RoboDK station: TRABAJO PRACTICO 7.rdk

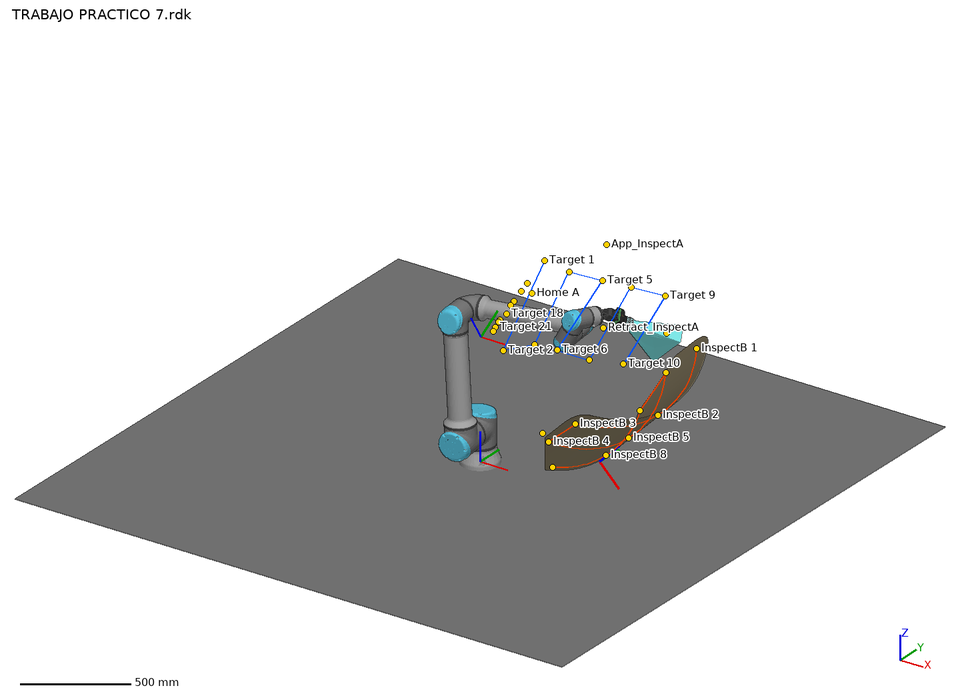
[picture v0: the station drawn from its stored meshes, robots at their saved joint values, targets as dots, program paths as lines]
Station TRABAJO PRACTICO 5 (saved by RoboDK 5.7.2). Poses are relative to the parent item; angles as X-Y-Z fixed-axis rotations.
Station parameters (name, value as stored): Palletizing Plugin
  - frame UR10e Base at (0, 0, 0) mm
    - robot UR10e: 6 axes, payload 10 kg, reach 1300 mm, repeatability 0.05 mm, weight 28.9 kg
        modified DH rows (alpha deg, a mm, theta deg, d mm): 0, 0, 0, 180.7; 90, 0, 180, 0; 0, 612.6, 0, 0; 0, 571.335, 0, 174.15; -90, 0, 0, 119.85; 90, 0, 180, 116.55
        joint limits [-360, -360, -360, -360, -360, -360] to [360, 360, 360, 360, 360, 360]; home [0, -90, -90, 0, 90, 0]; saved at [6.14, -86.815, -90.402, -30.486, 158.848, 109.654]
      - tool Camera 2, TCP at (0, -175.95, 321.06) mm, rotated rx 40 ry 0 rz 0 deg, size 215.7 x 276.1 x 372.4 mm
  - frame Frame Inspection A at (-380.72, 553.59, 295.24) mm, rotated rx 32.84 ry 0 rz 0 deg
    - object Inspection A at (0, 0, 0) mm, size 800 x 500 x 0 mm, geometry from Inspection A.step
    - folder TargetsA
    - target Target 1 (Cartesian target) at (79.2, 457.51, 5) mm, rotated rx -180 ry 0 rz 180 deg; joints [133.501, -90.589, -95.318, -17.151, 48.873, 195.641] of UR10e
    - target Target 2 (Cartesian target) at (141.75, -34.27, 5) mm, rotated rx 179.75 ry 0 rz 180 deg; joints [184.834, -41.161, -136.372, -107.963, 17.565, 286.215] of UR10e
    - target Target 3 (Cartesian target) at (270.26, 41.79, 5) mm, rotated rx 180 ry 0 rz 180 deg; joints [161.24, -38.764, -144.388, -40.681, 25.213, 220.978] of UR10e
    - target Target 4 (Cartesian target) at (224.75, 441.5, 5) mm, rotated rx -180 ry 0 rz 180 deg; joints [123.151, -84.661, -102.076, -13.507, 58.499, 190.907] of UR10e
    - target Target 5 (Cartesian target) at (403.61, 448.09, 5) mm, rotated rx -180 ry 0 rz 180 deg; joints [105.682, -83.563, -102.861, -11.357, 75.033, 184.735] of UR10e
    - target Target 6 (Cartesian target) at (390.7, 47.14, 5) mm, rotated rx 180 ry 0 rz 180 deg; joints [137.831, -39.235, -146.275, -19.19, 44.913, 198.041] of UR10e
    - target Target 7 (Cartesian target) at (568.48, 46.93, 5) mm, rotated rx -180 ry 0 rz 180 deg; joints [86.626, -56.24, -142.379, 1.432, 93.224, 179.004] of UR10e
    - target Target 8 (Cartesian target) at (554.74, 458.13, 5) mm, rotated rx -180 ry 0 rz 180 deg; joints [90.013, -86.994, -99.225, -10.94, 89.988, 180.004] of UR10e
    - target Target 9 (Cartesian target) at (750.45, 458.08, 25) mm, rotated rx 180 ry 0 rz 180 deg; joints [71.618, -93.897, -90.519, -13.607, 107.537, 174.401] of UR10e
    - target Target 10 (Cartesian target) at (750.21, 68.01, 25) mm, rotated rx 180 ry 0 rz 180 deg; joints [55.701, -74.55, -129.53, 3.586, 122.577, 168.622] of UR10e
    - target App_InspectA (Cartesian target) at (433.96, 543.11, 175.01) mm, rotated rx -172.24 ry 18.28 rz 174.82 deg; joints [115.29, -89.41, -72.94, -49.41, 49.41, 188.24] of UR10e
    - target Retract_InspectA (Cartesian target) at (750.21, 68.01, 315) mm, rotated rx 180 ry 0 rz -180 deg; joints [39.031, -62.165, -111.409, -32.544, 137.922, 160.003] of UR10e
    - target Home A (joint target) at (558.33, -45.25, 667.51) mm, rotated rx -180 ry 0 rz -180 deg; joints [90.932, -32.458, -85.483, -79.221, 89.109, 180.275] of UR10e
    - target Target 14 (Cartesian target) at (65.12, 323.89, 5) mm, rotated rx 180 ry 0 rz 179.79 deg; joints [142.957, -81.972, -110.313, -14.929, 40.175, 201.57] of UR10e
    - target Target 15 (Cartesian target) at (61.03, 276.19, 5) mm, rotated rx 180 ry 0 rz 179.79 deg; joints [146.894, -78.963, -115.197, -15.414, 36.711, 204.58] of UR10e
    - target Target 16 (Cartesian target) at (54.59, 218.09, 5) mm, rotated rx 180 ry 0 rz 179.79 deg; joints [152.333, -75.295, -120.754, -17.699, 32.077, 209.635] of UR10e
    - target Target 17 (Cartesian target) at (48.84, 192.68, 5) mm, rotated rx 180 ry 0 rz 179.79 deg; joints [155.072, -73.816, -122.904, -19.652, 29.834, 212.694] of UR10e
    - target Target 18 (Cartesian target) at (54.37, 146.46, 5) mm, rotated rx -180 ry -0.47 rz 179.79 deg; joints [159.377, -69.627, -127.627, -23.673, 26.763, 218.279] of UR10e
    - target Target 19 (Cartesian target) at (41.82, 108.93, 5) mm, rotated rx 180 ry 0 rz 179.79 deg; joints [164.318, -67.471, -129.772, -31.808, 22.992, 226.811] of UR10e
    - target Target 20 (Cartesian target) at (40.49, 96.72, 5) mm, rotated rx 180 ry 0 rz 179.79 deg; joints [165.792, -66.439, -130.582, -34.771, 22.053, 229.778] of UR10e
    - target Target 21 (Cartesian target) at (41.12, 65.11, 5) mm, rotated rx -180 ry 0 rz 179.79 deg; joints [169.618, -63.229, -132.561, -44.277, 19.903, 238.637] of UR10e
    - target Target 22 (Cartesian target) at (42.77, 42.7, 5) mm, rotated rx -180 ry 0 rz 179.79 deg; joints [172.451, -60.718, -133.61, -53.008, 18.646, 246.336] of UR10e
  - frame Frame Inspection B at (727.24, -100, 245.26) mm, rotated rx 0 ry 45.31 rz 0 deg
    - object Inspection B at (0, 0, 0) mm, size 202.5 x 1023.2 x 500 mm, geometry from Inspection B.step
    - target InspectB 1 (Cartesian target) at (-169.52, 507.12, 414.46) mm, rotated rx 90.86 ry 88.34 rz 129.57 deg; joints [15.023, -98.718, -87.565, -11.255, 155.215, 119.931] of UR10e
    - target InspectB 2 (Cartesian target) at (-6.3, 34.85, 422.21) mm, rotated rx 90 ry 88.73 rz 89.24 deg; joints [-2.551, -95.184, -85.812, -44.784, 131.035, 89.277] of UR10e
    - target InspectB 3 (Cartesian target) at (-170.32, -428.18, 402.32) mm, rotated rx 89.84 ry 89 rz 51.46 deg; joints [-17.421, -91.076, -80.259, -55.032, 103.875, 78.266] of UR10e
    - target InspectB 4 (Cartesian target) at (-180.94, -441.02, 219.27) mm, rotated rx 91.56 ry 89 rz 52.19 deg; joints [-22.212, -79.982, -102.696, -44.394, 106.19, 74.724] of UR10e
    - target InspectB 5 (Cartesian target) at (-6.33, 32.62, 194.61) mm, rotated rx 90 ry 89.2 rz 89.24 deg; joints [-3.525, -82.536, -114.24, -30.023, 131.7, 87.717] of UR10e
    - target InspectB 6 (Cartesian target) at (-168.47, 505.6, 180.05) mm, rotated rx 93.22 ry 89.38 rz 132.09 deg; joints [19.329, -87.442, -116.77, 8.038, 151.578, 120.916] of UR10e
    - target InspectB 7 (Cartesian target) at (-96.46, 396.52, 16.99) mm, rotated rx 90.7 ry 89.4 rz 119.27 deg; joints [17.027, -80.228, -135.951, 10.169, 144.428, 112.006] of UR10e
    - target InspectB 8 (Cartesian target) at (-6.25, 41.26, 15.39) mm, rotated rx 90.07 ry 89.47 rz 90.84 deg; joints [-4.974, -75.499, -133.485, -19.186, 134.195, 85.804] of UR10e
    - target InspectB 9 (Cartesian target) at (-88.51, -301.4, 19.49) mm, rotated rx 90.88 ry 89.53 rz 63.85 deg; joints [-21.86, -72.359, -126.788, -31.965, 117.705, 73.128] of UR10e
    - target App_InspectB (Cartesian target) at (-298.16, 404, 414.54) mm, rotated rx 90.86 ry 88.34 rz 129.57 deg; joints [7.716, -89.072, -88.225, -26.91, 162.055, 112.785] of UR10e
    - target Retract_InspectB (Cartesian target) at (-242.37, -222.92, 19.51) mm, rotated rx 90.88 ry 89.53 rz 63.85 deg; joints [-15.839, -53.956, -125.352, -49.575, 113.831, 78.249] of UR10e
  - frame World at (0, 0, 0) mm
    - object Floor at (0, 0, -7) mm, size 3000 x 3000 x 4.2 mm, geometry from Floor.step
  - folder InspectA
    - program GoHomeA (3 instructions, listed below)
    - program InspectA (12 instructions, listed below)
    - program MainInspectA (5 instructions, listed below)
    - program App_InspectA (3 instructions, listed below)
    - program Retract_InspectA (3 instructions, listed below)
  - folder InspectB
    - program InspectB (8 instructions, listed below)
    - program App_InspectB (3 instructions, listed below)
    - program Retract_InspectB (3 instructions, listed below)
    - program Main_InspectB (3 instructions, listed below)
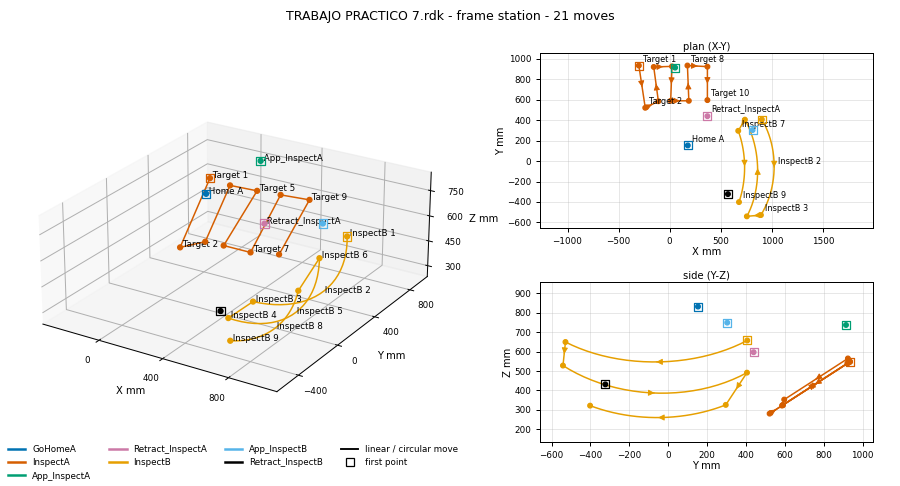
[picture p0: tool path of TRABAJO PRACTICO 7.rdk in frame station, 21 of 21 moves have a stored position in this frame; points joined in program order, loops and branches not executed]

--- program GoHomeA (robot UR10e) ---
  Est. Ref.: Frame Inspection A
  Est. herr: Camera 2
  MoveJ (Home A)

--- program InspectA (robot UR10e) ---
  Est. Ref.: Frame Inspection A
  Est. herr: Camera 2
  MoveJ (Target 1)
  MoveL (Target 2)
  MoveL (Target 3)
  MoveL (Target 4)
  MoveL (Target 5)
  MoveL (Target 6)
  MoveL (Target 7)
  MoveL (Target 8)
  MoveL (Target 9)
  MoveL (Target 10)

--- program MainInspectA (robot UR10e) ---
  Llamar GoHomeA
  Llamar App_InspectA
  Llamar InspectA
  Llamar Retract_InspectA
  Llamar GoHomeA

--- program App_InspectA (robot UR10e) ---
  Est. Ref.: Frame Inspection A
  Est. herr: Camera 2
  MoveJ (App_InspectA)

--- program Retract_InspectA (robot UR10e) ---
  Est. Ref.: Frame Inspection A
  Est. herr: Camera 2
  MoveL (Retract_InspectA)

--- program InspectB (robot UR10e) ---
  Est. Ref.: Frame Inspection B
  Est. herr: Camera 2
  MoveL (InspectB 1)
  MoveC (InspectB 2, InspectB 3)
  MoveL (InspectB 4)
  MoveC (InspectB 5, InspectB 6)
  MoveL (InspectB 7)
  MoveC (InspectB 8, InspectB 9)

--- program App_InspectB (robot UR10e) ---
  Est. Ref.: Frame Inspection B
  Est. herr: Camera 2
  MoveJ (App_InspectB)

--- program Retract_InspectB (robot UR10e) ---
  Est. Ref.: Frame Inspection B
  Est. herr: Camera 2
  MoveJ (Retract_InspectB)

--- program Main_InspectB (robot UR10e) ---
  Llamar App_InspectB
  Llamar Prog6
  Llamar Retract_InspectB
